(* Logix 5000 project; controller Latch_and_Unlatch Emulate 5570 rev 30.12; software revision 30.01 *)

TASK MainTask (continuous, watchdog 500 ms) : MainProgram

MODULES
   Local : Emulate 5570 (ICP 2, rev 30.12)
END_MODULES

PROGRAM MainProgram   (* main routine MainRoutine *)
VAR
   Motor : BOOL;
   PB1 : BOOL;
   PB2 : BOOL;
END_VAR

ROUTINE MainRoutine   (* ladder *)
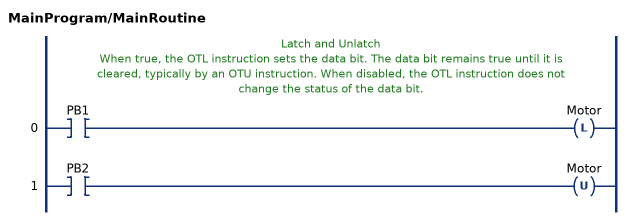
   // Latch and Unlatch
   // When true, the OTL instruction sets the data bit. The data bit remains true until it is cleared, typically by an OTU instruction. When disabled, the OTL instruction does not change the status of the data bit.
   0: XIC(PB1)OTL(Motor);
   1: XIC(PB2)OTU(Motor);
END_ROUTINE
END_PROGRAM
